ABB RAPID module: ModuleFab.mod

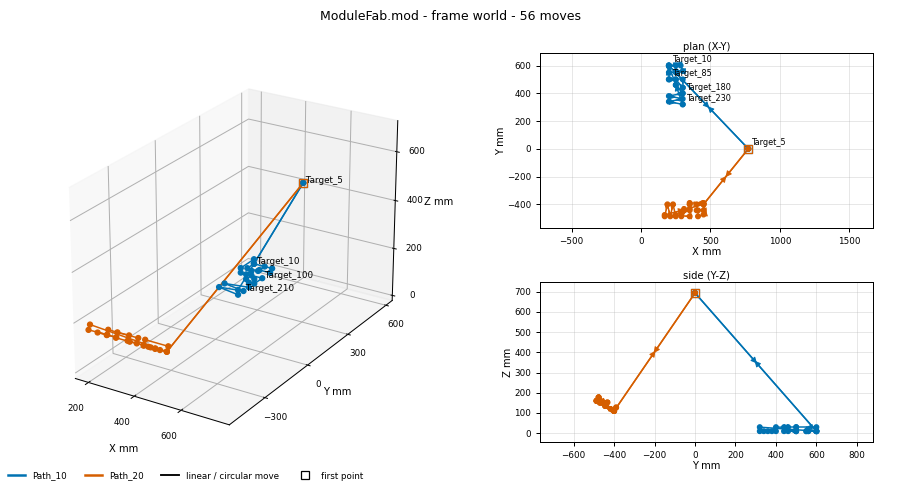
[picture p0: tool path of ModuleFab.mod in frame world, 56 of 56 moves have a stored position in this frame; points joined in program order, loops and branches not executed]
MODULE ModuleFab
    PERS tooldata Marker:=[TRUE,[[-0.917808,-1.75486,202.667],[0.812949,-0.58005,0.0419499,-0.0299318]],[0.2,[0,0,1],[1,0,0,0],0,0,0]];
    PERS wobjdata Cuadrante1:=[FALSE,TRUE,"",[[200,600,10],[1,0,0,0]],[[0,0,0],[1,0,0,0]]];
    PERS wobjdata Cuadrante2:=[FALSE,TRUE,"",[[450,-400,110],[0.683012702,-0.183012702,-0.183012702,-0.683012702]],[[0,0,0],[1,0,0,0]]];
    CONST robtarget Target_5:=[[-54.660161362,322.568528773,705.32582312],[0.5,-0.683012702,-0.5,-0.183012702],[0,0,0,0],[9E+09,9E+09,9E+09,9E+09,9E+09,9E+09]];
    CONST robtarget Target_10:=[[0.000029436,0.000002786,-0.00001954],[0,1,0,0],[0,0,0,0],[9E+09,9E+09,9E+09,9E+09,9E+09,9E+09]];
    CONST robtarget Target_20:=[[85.00007128,0.000056558,-0.000067404],[0.000000052,1,0.00000008,0.000000048],[0,-1,0,0],[9E+09,9E+09,9E+09,9E+09,9E+09,9E+09]];
    CONST robtarget Target_30:=[[100,-40,0],[0,1,0,0],[0,0,0,0],[9E+09,9E+09,9E+09,9E+09,9E+09,9E+09]];
    CONST robtarget Target_40:=[[49.999974739,-40.000167176,-0.000220434],[0.000000085,1,0.00000012,0.000000017],[0,0,0,0],[9E+09,9E+09,9E+09,9E+09,9E+09,9E+09]];
    CONST robtarget Target_50:=[[50.000010209,-0.000224541,-0.000250887],[0.000000134,1,0.000000203,0.000000033],[0,0,0,0],[9E+09,9E+09,9E+09,9E+09,9E+09,9E+09]];
    CONST robtarget Target_60:=[[50.000025112,-50.000553987,-0.000343463],[-0.000000118,1,0.00000012,0.000000003],[0,-1,0,0],[9E+09,9E+09,9E+09,9E+09,9E+09,9E+09]];
    CONST robtarget Target_70:=[[-0.000006592,-50.000589308,-0.000400325],[0.000000139,1,0.000000133,0.000000007],[0,0,0,0],[9E+09,9E+09,9E+09,9E+09,9E+09,9E+09]];
    CONST robtarget Target_75:=[[-0.000022603,-0.000576441,-0.000529581],[-0.000000124,1,0.000000261,0.000000006],[0,-1,0,0],[9E+09,9E+09,9E+09,9E+09,9E+09,9E+09]];
    CONST robtarget Target_80:=[[0,-0.001,20],[0,1,0,0],[0,0,0,0],[9E+09,9E+09,9E+09,9E+09,9E+09,9E+09]];
    CONST robtarget Target_85:=[[0,-100.001,20],[0,1,0,0],[0,0,0,0],[9E+09,9E+09,9E+09,9E+09,9E+09,9E+09]];
    CONST robtarget Target_90:=[[0.000025927,-100.000700186,-0.000677472],[-0.000000107,1,0.00000022,-0.000000007],[0,-1,0,0],[9E+09,9E+09,9E+09,9E+09,9E+09,9E+09]];
    CONST robtarget Target_100:=[[99.999989388,-100.000679508,-0.000800598],[-0.000000117,1,0.000000284,0.000000009],[0,-1,0,0],[9E+09,9E+09,9E+09,9E+09,9E+09,9E+09]];
    CONST robtarget Target_110:=[[100.000005029,-160.000691199,-0.000896846],[-0.000000109,1,0.000000357,0.000000012],[0,-1,0,0],[9E+09,9E+09,9E+09,9E+09,9E+09,9E+09]];
    CONST robtarget Target_120:=[[100.00000373,-160.000694861,19.999066559],[-0.000000108,1,0.000000367,0.000000014],[0,-1,0,0],[9E+09,9E+09,9E+09,9E+09,9E+09,9E+09]];
    CONST robtarget Target_130:=[[49.999968629,-100.00068441,19.998940551],[0.00000011,1,0.000000227,0.000000029],[0,0,0,0],[9E+09,9E+09,9E+09,9E+09,9E+09,9E+09]];
    CONST robtarget Target_140:=[[50.000028108,-100.000699853,-0.00110166],[0.000000088,1,0.000000216,0.000000026],[0,0,0,0],[9E+09,9E+09,9E+09,9E+09,9E+09,9E+09]];
    CONST robtarget Target_150:=[[50.000019247,-140.000721368,-0.001141499],[0.000000091,1,0.000000183,0.000000028],[0,0,0,0],[9E+09,9E+09,9E+09,9E+09,9E+09,9E+09]];
    CONST robtarget Target_160:=[[50.000021567,-140.000727631,19.998828298],[0.000000102,1,0.000000189,0.000000033],[0,0,0,0],[9E+09,9E+09,9E+09,9E+09,9E+09,9E+09]];
    CONST robtarget Target_180:=[[100.000022516,-200.000718847,19.998012068],[-0.000000105,1,0.000000139,0.000000072],[0,-1,0,0],[9E+09,9E+09,9E+09,9E+09,9E+09,9E+09]];
    CONST robtarget Target_190:=[[100.000012664,-200.000722966,-0.002015141],[-0.000000111,1,0.000000147,0.000000064],[0,-1,0,0],[9E+09,9E+09,9E+09,9E+09,9E+09,9E+09]];
    CONST robtarget Target_200:=[[0.000004659,-220.000687419,-0.002157373],[-0.00000012,1,0.0000001,0.000000078],[0,-1,0,0],[9E+09,9E+09,9E+09,9E+09,9E+09,9E+09]];
    CONST robtarget Target_210:=[[100.000008139,-240.000689264,-0.002308121],[-0.000000136,1,0.000000073,0.000000105],[0,-1,0,0],[9E+09,9E+09,9E+09,9E+09,9E+09,9E+09]];
    CONST robtarget Target_220:=[[0.000105568,-260.000728838,-0.0024296],[0.000000037,1,-0.000000001,0.000000182],[0,-1,0,0],[9E+09,9E+09,9E+09,9E+09,9E+09,9E+09]];
    CONST robtarget Target_230:=[[100.00010508,-280.000701552,-0.002614694],[-0.000000019,1,-0.000000044,0.000000209],[0,-1,0,0],[9E+09,9E+09,9E+09,9E+09,9E+09,9E+09]];
    CONST robtarget Target_240:=[[100.000114302,-280.00069038,19.997361362],[-0.000000031,1,-0.000000041,0.000000218],[0,-1,0,0],[9E+09,9E+09,9E+09,9E+09,9E+09,9E+09]];
    CONST robtarget Target_250:=[[0.000008509,0.000003577,-0.00001118],[0.000000006,1,0,-0.000000002],[0,0,0,0],[9E+09,9E+09,9E+09,9E+09,9E+09,9E+09]];
    CONST robtarget Target_260:=[[-54.660161362,322.568528773,705.32582312],[0.5,-0.683012702,-0.5,-0.183012702],[0,0,0,0],[9E+09,9E+09,9E+09,9E+09,9E+09,9E+09]];

    PROC main10()
        Path_10;
        Path_20;
    ENDPROC
    PROC Path_10()
        MoveL Target_5,v200,z10,Marker\WObj:=Cuadrante2;
        MoveL Target_10,v200,z10,Marker\WObj:=Cuadrante1;
        MoveL Target_20,v200,z10,Marker\WObj:=Cuadrante1;
        MoveL Target_30,v200,z10,Marker\WObj:=Cuadrante1;
        MoveL Target_40,v200,z10,Marker\WObj:=Cuadrante1;
        MoveL Target_50,v200,z10,Marker\WObj:=Cuadrante1;
        MoveL Target_60,v200,z10,Marker\WObj:=Cuadrante1;
        MoveL Target_70,v200,z10,Marker\WObj:=Cuadrante1;
        MoveL Target_75,v200,z10,Marker\WObj:=Cuadrante1;
        MoveL Target_80,v200,z10,Marker\WObj:=Cuadrante1;
        MoveL Target_85,v200,z10,Marker\WObj:=Cuadrante1;
        MoveL Target_90,v200,z10,Marker\WObj:=Cuadrante1;
        MoveL Target_100,v200,z10,Marker\WObj:=Cuadrante1;
        MoveL Target_110,v200,z10,Marker\WObj:=Cuadrante1;
        MoveL Target_120,v200,z10,Marker\WObj:=Cuadrante1;
        MoveL Target_130,v200,z10,Marker\WObj:=Cuadrante1;
        MoveL Target_140,v200,z10,Marker\WObj:=Cuadrante1;
        MoveL Target_150,v200,z10,Marker\WObj:=Cuadrante1;
        MoveL Target_160,v200,z10,Marker\WObj:=Cuadrante1;
        MoveL Target_180,v200,z10,Marker\WObj:=Cuadrante1;
        MoveL Target_190,v200,z10,Marker\WObj:=Cuadrante1;
        MoveL Target_200,v200,z10,Marker\WObj:=Cuadrante1;
        MoveL Target_210,v200,z10,Marker\WObj:=Cuadrante1;
        MoveL Target_220,v200,z10,Marker\WObj:=Cuadrante1;
        MoveL Target_230,v200,z10,Marker\WObj:=Cuadrante1;
        MoveL Target_240,v200,z10,Marker\WObj:=Cuadrante1;
        MoveL Target_250,v200,z10,Marker\WObj:=Cuadrante1;
        MoveL Target_260,v200,z10,Marker\WObj:=Cuadrante2;
    ENDPROC
    PROC Path_20()
        MoveL Target_5,v200,z10,Marker\WObj:=Cuadrante2;
        MoveL Target_10,v200,z10,Marker\WObj:=Cuadrante2;
        MoveL Target_20,v200,z10,Marker\WObj:=Cuadrante2;
        MoveL Target_30,v200,z10,Marker\WObj:=Cuadrante2;
        MoveL Target_40,v200,z10,Marker\WObj:=Cuadrante2;
        MoveL Target_50,v200,z10,Marker\WObj:=Cuadrante2;
        MoveL Target_60,v200,z10,Marker\WObj:=Cuadrante2;
        MoveL Target_70,v200,z10,Marker\WObj:=Cuadrante2;
        MoveL Target_75,v200,z10,Marker\WObj:=Cuadrante2;
        MoveL Target_80,v200,z10,Marker\WObj:=Cuadrante2;
        MoveL Target_85,v200,z10,Marker\WObj:=Cuadrante2;
        MoveL Target_90,v200,z10,Marker\WObj:=Cuadrante2;
        MoveL Target_100,v200,z10,Marker\WObj:=Cuadrante2;
        MoveL Target_110,v200,z10,Marker\WObj:=Cuadrante2;
        MoveL Target_120,v200,z10,Marker\WObj:=Cuadrante2;
        MoveL Target_130,v200,z10,Marker\WObj:=Cuadrante2;
        MoveL Target_140,v200,z10,Marker\WObj:=Cuadrante2;
        MoveL Target_150,v200,z10,Marker\WObj:=Cuadrante2;
        MoveL Target_160,v200,z10,Marker\WObj:=Cuadrante2;
        MoveL Target_180,v200,z10,Marker\WObj:=Cuadrante2;
        MoveL Target_190,v200,z10,Marker\WObj:=Cuadrante2;
        MoveL Target_200,v200,z10,Marker\WObj:=Cuadrante2;
        MoveL Target_210,v200,z10,Marker\WObj:=Cuadrante2;
        MoveL Target_220,v200,z10,Marker\WObj:=Cuadrante2;
        MoveL Target_230,v200,z10,Marker\WObj:=Cuadrante2;
        MoveL Target_240,v200,z10,Marker\WObj:=Cuadrante2;
        MoveL Target_250,v200,z10,Marker\WObj:=Cuadrante2;
        MoveL Target_260,v200,z10,Marker\WObj:=Cuadrante2;
    ENDPROC
ENDMODULE
